IF (ipTcComObj=0) THEN
  GetObjPara := Tc2_System.E_HRESULTAdsErr.NOINTERFACE;
END_IF

IF (SUCCEEDED(GetObjPara)) THEN
  GetObjPara := ipTcComObj.TcGetObjPara(pid:=pid,nData,pData,0);
END_IF
END_METHOD

{attribute 'object_name' := 'Init'}
METHOD PROTECTED Init : HRESULT
VAR_INPUT
	oid: OTCID;
END_VAR

// preinitialize variables
memset(ADR(moduleClsId),0,SIZEOF(moduleClsId));
bClassIdVerified := FALSE;
hResult := Tc2_System.E_HRESULTAdsErr.HRESULT_ADS_NOERROR;

// get object server
IF (ipObjSrv=0) THEN
  hResult := FW_ObjMgr_GetObjectServer(_AppInfo.ObjId,ADR(ipObjSrv));
END_IF

// try to get object interfaces
IF (SUCCEEDED(hresult)) THEN
  QueryTcComInterface(hResult,oid);
END_IF

// verify class id
IF (SUCCEEDED(hresult)) THEN
  hresult := VerifyClassId();
END_IF

// query interfaces, if the current state is higher than INIT
IF (SUCCEEDED(hresult) AND State>TCOM_STATE.TCOM_STATE_INIT) THEN
  QueryObjInterfaces(hResult);
END_IF

// return value
Init := hresult;
END_METHOD

{attribute 'object_name' := 'InitObjName'}
METHOD PRIVATE InitObjName
VAR_INPUT
	hr: REFERENCE TO HRESULT;
END_VAR
VAR
	objectName: STRING(255) := 'TempContr_PlcRtFbInstance';
	oid: OTCID;
END_VAR

IF (SUCCEEDED(hr)) THEN
  hr := ipTcComObj.TcGetObjectId(oid);
END_IF

IF (SUCCEEDED(hr) and bDynInstance) THEN
  objectName := TC2_STANDARD.CONCAT(objectName,'_');
  objectName := TC2_STANDARD.CONCAT(objectName,UDINT_TO_STRING(oid));
  hr := ipTcComObj.TcSetObjectName(ADR(objectName));
END_IF
END_METHOD

{attribute 'object_name' := 'Internal_SetObjState'}
METHOD PROTECTED Internal_SetObjState
VAR_INPUT
	hr: REFERENCE TO HRESULT;
	nextState: TCOM_STATE;
END_VAR

// verify class id
IF (SUCCEEDED(hr)) THEN
  hr := VerifyClassId();
END_IF

// switch object state
IF (SUCCEEDED(hr) AND nextState>=TCOM_STATE_INIT) THEN
  IF (ipTcComObj=0) THEN
    hr := Tc2_System.E_HRESULTAdsErr.NOINTERFACE;
  END_IF
  IF (ipObjSrv=0) THEN
    hr := Tc2_System.E_HRESULTAdsErr.NOINTERFACE;
  END_IF
  IF (SUCCEEDED(hr)) THEN
    hr := ipTcComObj.TcSetObjState(nextState,ipObjSrv,pInitData);
  END_IF
END_IF
END_METHOD

{attribute 'object_name' := 'QueryObjInterface'}
METHOD PRIVATE QueryObjInterface
VAR_INPUT
	hr: REFERENCE TO HRESULT;
	iid: REFERENCE TO IID;
	pipItf: POINTER TO ITcUnknown;
END_VAR
VAR CONSTANT
	pNull: PVOID := 0;
END_VAR

IF (SUCCEEDED(hr)) THEN
  IF (ipTcComObj=0) THEN
    hr := Tc2_System.E_HRESULTAdsErr.NOINTERFACE;
  ELSIF (pipItf^=ULINT_TO_DWORD(pNull)) THEN
    hr := ipTcComObj.TcQueryInterface(iid:= iid, pipItf:=pipItf);
  END_IF
END_IF
END_METHOD

{attribute 'object_name' := 'QueryObjInterfaces'}
METHOD PRIVATE QueryObjInterfaces
VAR_INPUT
	hr: REFERENCE TO HRESULT;
END_VAR

IF(State<TCOM_STATE_PREOP)THEN
  hr := Tc2_System.E_HRESULTAdsErr.INVALIDSTATE;
END_IF

//cyclic interface
QueryObjInterface(hr,IID_ITCCYCLIC,ADR(ipTcCyclic));
//post cyclic interface
QueryObjInterface(hr,IID_ITCPOSTCYCLIC,ADR(ipTcPostCyclic));
//adi interface
QueryObjInterface(hr,IID_ITcADI,ADR(ipTcAdi));
END_METHOD

{attribute 'object_name' := 'QueryTcComInterface'}
METHOD PRIVATE QueryTcComInterface
VAR_INPUT
	hr: REFERENCE TO HRESULT;
	oid: OTCID;
END_VAR

IF (ipObjSrv=0) THEN
  hr := Tc2_System.E_HRESULTAdsErr.NOINTERFACE;
END_IF

IF (SUCCEEDED(hr) AND ipTcComObj=0) THEN
  bDynInstance := FALSE;
  IF(oid>0) THEN
    // query interface of existing object
    hr := ipObjSrv.TcQueryObjectInterface(oid,IID_ITComObject,ADR(ipTcComObj));
  ELSE
    // create new instance and get the object interface
    hr := ipObjSrv.TcCreateInstance(assignedClsId,IID_ITComObject,ADR(ipTcComObj));
    IF (SUCCEEDED(hr)) THEN
      bDynInstance := TRUE;
      hr := ipTcComObj.TcSetObjectId(OTCID_CreateNewId);
    END_IF
  END_IF
  IF (SUCCEEDED(hr)) THEN
    eInitialObjState := State;
  END_IF
END_IF
END_METHOD

{attribute 'object_name' := 'ReadModuleClassId'}
METHOD PRIVATE ReadModuleClassId : HRESULT
VAR
	emptyClsId: CLSID;
END_VAR
memset(ADR(emptyClsId),0,SIZEOF(emptyClsId));
IF (memcmp(ADR(moduleClsId),ADR(emptyClsId),SIZEOF(moduleClsId))=0) THEN
  IF (ipTcComObj=0) THEN
    ReadModuleClassId := Tc2_System.E_HRESULTAdsErr.NOINTERFACE;
  END_IF

  //objectClsId := clsid;
  IF (SUCCEEDED(ReadModuleClassId)) THEN
    ReadModuleClassId := ipTcComObj.GetClassId(moduleClsId);
  END_IF
END_IF
END_METHOD

{attribute 'object_name' := 'ReleaseImagePtrs'}
METHOD PRIVATE ReleaseImagePtrs : HRESULT
VAR
	nDaIdx: UDINT;
	pCurDataArea: POINTER TO ST_TcMatSimObjectDataAreaInfo;
END_VAR

IF (ipTcAdi=0) THEN
  ReleaseImagePtrs := Tc2_System.E_HRESULTAdsErr.NOINTERFACE;
END_IF

IF (SUCCEEDED(ReleaseImagePtrs) AND pDataAreas<>0) THEN
  // release pointers to the simulink module process images
  FOR nDaIdx:=0 TO nDataAreas-1 DO
    pCurDataArea := pDataAreas + nDaIdx*SIZEOF(ST_TcMatSimObjectDataAreaInfo);

    IF (pCurDataArea^.pModuleProcImg<>0) THEN
      ipTcAdi.ReleaseImagePtr(pData:=pCurDataArea^.pModuleProcImg);
      pCurDataArea^.pModuleProcImg := 0;
    END_IF
  END_FOR
END_IF
END_METHOD

{attribute 'object_name' := 'ReleaseObjInterfaces'}
METHOD PRIVATE ReleaseObjInterfaces : HRESULT

// release interface pointers
IF (ipTcCyclic<>0) THEN
  ipTcCyclic.TcRelease();
  ipTcCyclic := 0;
END_IF
IF (ipTcPostCyclic<>0) THEN
  ipTcPostCyclic.TcRelease();
  ipTcPostCyclic := 0;
END_IF
IF (ipTcAdi<>0) THEN
  ipTcAdi.TcRelease();
  ipTcAdi := 0;
END_IF
END_METHOD

{attribute 'object_name' := 'ReleaseTcComInterface'}
METHOD PRIVATE ReleaseTcComInterface : HRESULT
VAR
	nStateChangeCnt: DINT := 0;
END_VAR

IF (ipTcComObj<>0) THEN
  WHILE (State>eInitialObjState AND nStateChangeCnt<1000) DO
    State := eInitialObjState;
    nStateChangeCnt := nStateChangeCnt+1;
  END_WHILE
  ReleaseObjInterfaces();
  IF (bDynInstance) THEN
    ReleaseTcComInterface := TC3_MODULE.FW_ObjMgr_DeleteInstance(ADR(ipTcComObj));
  ELSE
    ipTcComObj.TcRelease();
  END_IF
  ipTcComObj := 0;
END_IF
END_METHOD

{attribute 'object_name' := 'ResetHresult'}
METHOD ResetHresult
hResult := S_OK;
END_METHOD

{attribute 'object_name' := 'SaveOnlineParametersForInit'}
METHOD SaveOnlineParametersForInit : HRESULT
VAR
	idx: UINT;
	pInitElemHdr: POINTER TO TComInitDataElmHdr;
	pData: PVOID;
	nData: UDINT;
END_VAR
VAR CONSTANT
	nInitDataAlignment: UDINT := 4;
END_VAR
IF (pInitData<>0) THEN
  pInitElemHdr := pInitData + SIZEOF(pInitData^);
  FOR idx:=1 TO pInitData^.uiElmCnt DO
    pData := pInitElemHdr + ULINT_TO_DWORD(SIZEOF(pInitElemHdr^));
    nData := pInitElemHdr^.cbData;
    SaveOnlineParametersForInit := GetObjPara(pInitElemHdr^.indexOffset,nData,pData);
    IF (FAILED(SaveOnlineParametersForInit)) THEN
      RETURN;
    END_IF
    pInitElemHdr := pData + (nInitDataAlignment*((nData + nInitDataAlignment - 1)/nInitDataAlignment));
  END_FOR
ELSE
	SaveOnlineParametersForInit := Tc2_System.E_HRESULTAdsErr.NOTINIT;
END_IF
END_METHOD


METHOD PUBLIC SetDataAreaInfo
VAR_INPUT
  pDataAreas: POINTER TO ST_TcMatSimObjectDataAreaInfo;
  nDataAreas: UDINT;
END_VAR

THIS^.nDataAreas := nDataAreas;
THIS^.pDataAreas := pDataAreas;
END_METHOD


METHOD PUBLIC SetInitDataInfo
VAR_INPUT
  pInitData : POINTER TO TComInitDataHdr;
END_VAR
this^.pInitData := pInitData;
END_METHOD

{attribute 'object_name' := 'SetObjPara'}
METHOD SetObjPara : HRESULT
VAR_INPUT
	pid: PTCID;
	nData: UDINT;
	pData: PVOID;
END_VAR

IF (ipTcComObj=0) THEN
  SetObjPara := Tc2_System.E_HRESULTAdsErr.NOINTERFACE;
END_IF

IF (SUCCEEDED(SetObjPara)) THEN
  SetObjPara := ipTcComObj.TcSetObjPara(pid:=pid,nData,pData,0);
END_IF
END_METHOD

{attribute 'object_name' := 'SetObjState'}
METHOD SetObjState : HRESULT
VAR_INPUT
	finalState: TCOM_STATE;
END_VAR
VAR
	bShiftUp: BOOL;
	bShiftDown: BOOL;
	currentState: TCOM_STATE;
END_VAR

currentState := State;

bShiftUp := finalState>currentState;
bShiftDown := finalState<currentState;

// do not switch up on error
IF (FAILED(hresult)) THEN
  bShiftUp := FALSE;
END_IF
// reset existing error on switching down
IF (bShiftDown) THEN
  ResetHresult();
END_IF

// prepared state switch
CASE currentState OF
  TCOM_STATE_INIT:
    IF(bShiftUp) THEN
      QueryTcComInterface(hResult,0);
      Internal_SetObjState(hResult,TCOM_STATE.TCOM_STATE_PREOP);
      InitObjName(hResult);
    END_IF

  TCOM_STATE_PREOP:
    IF(bShiftUp) THEN
      Internal_SetObjState(hResult,TCOM_STATE.TCOM_STATE_SAFEOP);
      QueryObjInterfaces(hResult);
    ELSIF (bShiftDown) THEN
      Internal_SetObjState(hResult,TCOM_STATE.TCOM_STATE_INIT);
    END_IF

  TCOM_STATE_SAFEOP:
    IF(bShiftUp) THEN
      Internal_SetObjState(hResult,TCOM_STATE.TCOM_STATE_OP);
      QueryObjInterfaces(hResult);
    ELSIF (bShiftDown) THEN
      Internal_SetObjState(hResult,TCOM_STATE.TCOM_STATE_PREOP);
      ReleaseObjInterfaces();
    END_IF


  TCOM_STATE_OP:
    IF (bShiftDown) THEN
      Internal_SetObjState(hResult,TCOM_STATE.TCOM_STATE_SAFEOP);
    END_IF
END_CASE

SetObjState := hResult;
END_METHOD

PROPERTY State : TCOM_STATE
GET
VAR
	hr: HRESULT := S_OK;
	eObjState: TCOM_STATE;
END_VAR

IF (ipTcComObj<>0) THEN
  hr := ipTcComObj.TcGetObjState(ADR(eObjState));
IF (FAILED(hr)) THEN
  eObjState := TCOM_STATE.TCOM_STATE_INIT;
END_IF
ELSE
  eObjState := TCOM_STATE.TCOM_STATE_INIT;
END_IF
State := eObjState;
END_GET
SET
SetObjState(State);
END_SET
END_PROPERTY

{attribute 'object_name' := 'VerifyClassId'}
METHOD PRIVATE VerifyClassId : HRESULT
VAR
	emptyClsId: CLSID;
END_VAR
memset(ADR(emptyClsId),0,SIZEOF(emptyClsId));
IF (bClassIdVerified) THEN
  // class ID was already verified
  VerifyClassId := Tc2_System.E_HRESULTAdsErr.HRESULT_ADS_NOERROR;
ELSIF (memcmp(ADR(assignedClsId),ADR(emptyClsId),SIZEOF(assignedClsId))=0) THEN
  // skip class ID verification if no assignedClsId specified
  VerifyClassId := Tc2_System.E_HRESULTAdsErr.HRESULT_ADS_NOERROR;
ELSE
  // verify class ID
  VerifyClassId := ReadModuleClassId();

  IF (SUCCEEDED(VerifyClassId)) THEN
    IF (memcmp(ADR(assignedClsId),ADR(moduleClsId),SIZEOF(assignedClsId))<>0) THEN
     VerifyClassId := Tc2_System.E_HRESULTAdsErr.INVALIDCLSID;
    END_IF
  END_IF
  bClassIdVerified := SUCCEEDED(VerifyClassId);
END_IF
END_METHOD

END_FUNCTION_BLOCK

// ---- GlobalTextList.TcGTLO
TEXTLIST GlobalTextList
  145 = ' %.2f'
  175 = ' realState=%.3f'
  165 = ' t_Interval=%.2f'
  167 = ' t_Interval=%.3f'
  169 = ' t_Interval=%.4f'
  168 = ' t_Interval=%.5f'
  143 = '%.2f'
  179 = '1'
  81 = 'Axis10_Back'
  82 = 'Axis10_Home'
  117 = 'Axis10_Move'
  11 = 'Axis10_Power'
  83 = 'Axis11_Back'
  84 = 'Axis11_Home'
  118 = 'Axis11_Move'
  12 = 'Axis11_Power'
  85 = 'Axis12_Back'
  86 = 'Axis12_Home'
  119 = 'Axis12_Move'
  13 = 'Axis12_Power'
  87 = 'Axis13_Back'
  88 = 'Axis13_Home'
  120 = 'Axis13_Move'
  14 = 'Axis13_Power'
  89 = 'Axis14_Back'
  90 = 'Axis14_Home'
  121 = 'Axis14_Move'
  15 = 'Axis14_Power'
  91 = 'Axis15_Back'
  92 = 'Axis15_Home'
  122 = 'Axis15_Move'
  16 = 'Axis15_Power'
  93 = 'Axis16_Back'
  94 = 'Axis16_Home'
  123 = 'Axis16_Move'
  17 = 'Axis16_Power'
  95 = 'Axis17_Back'
  96 = 'Axis17_Home'
  124 = 'Axis17_Move'
  18 = 'Axis17_Power'
  97 = 'Axis18_Back'
  98 = 'Axis18_Home'
  125 = 'Axis18_Move'
  19 = 'Axis18_Power'
  62 = 'Axis1_Back'
  64 = 'Axis1_Home'
  63 = 'Axis1_Home_Set'
  106 = 'Axis1_M'
  108 = 'Axis1_Move'
  2 = 'Axis1_Power'
  65 = 'Axis2_Back'
  66 = 'Axis2_Home'
  109 = 'Axis2_Move'
  3 = 'Axis2_Power'
  67 = 'Axis3_Back'
  68 = 'Axis3_Home'
  110 = 'Axis3_Move'
  4 = 'Axis3_Power'
  69 = 'Axis4_Back'
  70 = 'Axis4_Home'
  111 = 'Axis4_Move'
  5 = 'Axis4_Power'
  71 = 'Axis5_Back'
  72 = 'Axis5_Home'
  112 = 'Axis5_Move'
  6 = 'Axis5_Power'
  73 = 'Axis6_Back'
  74 = 'Axis6_Home'
  113 = 'Axis6_Move'
  7 = 'Axis6_Power'
  75 = 'Axis7_Back'
  76 = 'Axis7_Home'
  114 = 'Axis7_Move'
  8 = 'Axis7_Power'
  77 = 'Axis8_Back'
  78 = 'Axis8_Home'
  115 = 'Axis8_Move'
  9 = 'Axis8_Power'
  79 = 'Axis9_Back'
  80 = 'Axis9_Home'
  116 = 'Axis9_Move'
  10 = 'Axis9_Power'
  56 = 'Axis_ActPostion[INDEX]'
  60 = 'Back'
  174 = 'Botton For Step'
  57 = 'Current_Turque_Value[INDEX]'
  39 = 'Driver10_Reset'
  40 = 'Driver11_Reset'
  41 = 'Driver12_Reset'
  42 = 'Driver13_Reset'
  43 = 'Driver14_Reset'
  44 = 'Driver15_Reset'
  45 = 'Driver16_Reset'
  46 = 'Driver17_Reset'
  47 = 'Driver18_Reset'
  30 = 'Driver1_Reset'
  31 = 'Driver2_Reset'
  32 = 'Driver3_Reset'
  33 = 'Driver4_Reset'
  34 = 'Driver5_Reset'
  35 = 'Driver6_Reset'
  36 = 'Driver7_Reset'
  37 = 'Driver8_Reset'
  38 = 'Driver9_Reset'
  127 = 'Error & Reset'
  126 = 'Error&Reset'
  151 = 'Exsetopint_Enable'
  152 = 'Exsetopint_On'
  141 = 'Exsetpoint_Exectue'
  23 = 'Home'
  59 = 'Home_Execute'
  61 = 'Home_Set'
  131 = 'Leg1_Home'
  181 = 'Leg21'
  132 = 'Leg2_Home'
  133 = 'Leg3_Home'
  134 = 'Leg4_Home'
  135 = 'Leg5_Home'
  136 = 'Leg6_Home'
  180 = 'Leg_1'
  186 = 'Leg_16'
  182 = 'Leg_2'
  183 = 'Leg_3'
  184 = 'Leg_4'
  185 = 'Leg_5'
  187 = 'Leg_6'
  177 = 'Model_Position[INDEX]'
  130 = 'Move & Stand'
  107 = 'MoveAbsoluteDone[INDEX]'
  129 = 'Move_Execute'
  53 = 'Power'
  20 = 'Power_Execute'
  188 = 'RealState=%.3f'
  29 = 'Reset'
  49 = 'Reset_Execute'
  26 = 'Robot_Error'
  101 = 'Robot_Home_Set'
  0 = 'Robot_Power'
  48 = 'Robot_Reset'
  128 = 'Robot_Stand_Execute'
  99 = 'Robot_Start_Back'
  100 = 'sadad'
  166 = 'Simulink_Move'
  176 = 'State=%.3f'
  189 = 'Step_Test'
  147 = 't=%.2f'
  170 = 't=%.3f'
  171 = 'Touch_Signal'
  178 = 'Touch_Signal(模型中腿编号)'
  172 = 'Touch_Signal_1'
  173 = 'Touch_Signal_Change'
  144 = 'T_ALL = %.2f'
  158 = 't_Interval=%.2f'
  22 = '切换视图'
  157 = '取样时间间隔 t_Interval'
  160 = '取样时间间隔 t_Interval(ms)'
  161 = '取样时间间隔 t_Interval(s)'
  159 = '取样时间间隔 t_Interval/ms'
  139 = '可以用来整体机器人运动'
  140 = '可以用来整体机器人进行Simulink模型验证'
  104 = '可以用来给单个四缸伸长或者是整体机器人站立'
  28 = '可以用来给单个电机或者是整体机器人上电'
  55 = '可以用来给单个电机或者是整体机器人找零'
  103 = '可以用来给单个电机或者是整体机器人站立'
  52 = '可以用来错误时给单个电机或者是整体机器人进行驱动重置'
  24 = '否'
  149 = '开始输入轨迹'
  156 = '当前取样时间 t'
  163 = '当前取样时间 t(s)'
  25 = '是'
  148 = '是否开始输入轨迹'
  21 = '是否进行上电操作'
  58 = '是否进行找零操作'
  1 = '是否进行整机操作'
  142 = '是否进行运动操作'
  50 = '是否进行驱动重置'
  138 = '本界面为电机Sumulink模型运动程序：'
  137 = '本界面为电机Sumulink程序：'
  27 = '本界面为电机上电程序：'
  102 = '本界面为电机伸长/机器人站立程序：'
  54 = '本界面为电机找零程序：'
  105 = '本界面为电机绝对运动/机器人站立程序：'
  51 = '本界面为驱动重置程序：'
  154 = '输入运动总时长 T_ALL'
  162 = '输入运动总时长 T_ALL(s)'
  150 = '运动当前时间 t'
  164 = '运动当前时间 t(s)'
  146 = '运动总时长 T_ALL'
  155 = '运动时间间隔 t'
  153 = '运动终止信号'
END_TEXTLIST

// ---- VISUs/Visu_Home.TcVIS
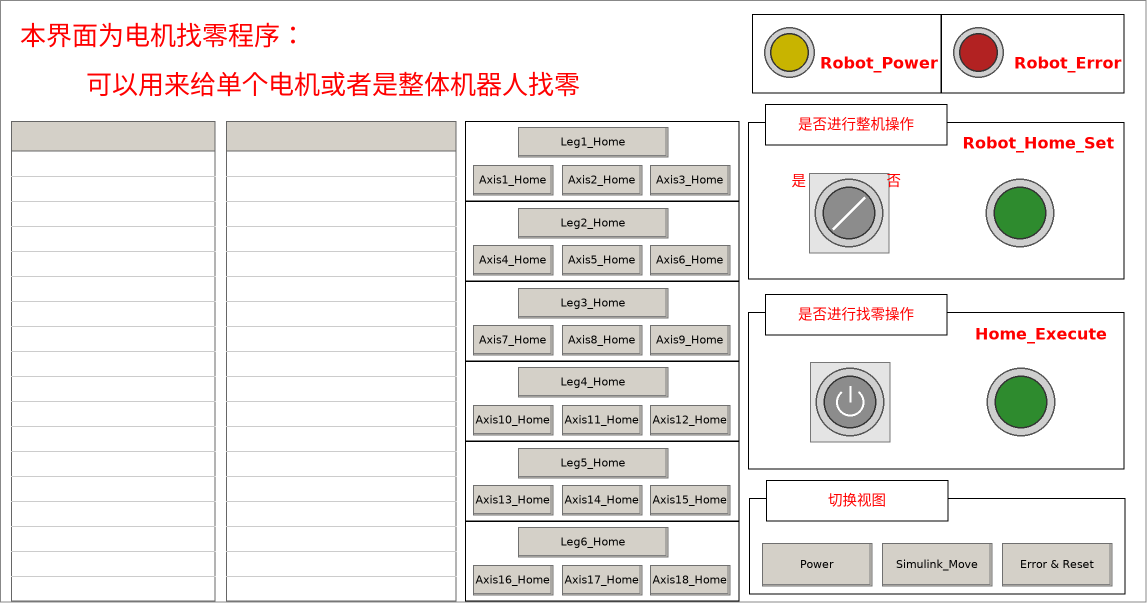
VISUALIZATION Visu_Home  // 1147x603
    Rectangle (752,14 189x79)
    Rectangle (748,312 376x157)
    Label (964,318 154x32), "Home_Execute"
    Rectangle (765,294 182x41), "是否进行找零操作"
    Lamp1 (981,362 80x80), variable: MAIN.Home_Execute, style: Lamp-Lamp1-Green
    PowerSwitch (810,362 80x80), variable: MAIN.Home_Execute, behaviour: TOGGLE, style: Switch-PowerSwitch-Gray
    Rectangle (941,14 183x79)
    Lamp1 (948,23 61x59), variable: MAIN.Robot_Error, style: Lamp-Lamp1-Red
    Label (991,47 154x32), "Robot_Error"
    Label (17,15 365x42), "本界面为电机找零程序："
    Label (83,64 874x42), "可以用来给单个电机或者是整体机器人找零"
    Table (11,121 204x480), data array: MAIN.Axis_ActPostion
        p3854506369: MAIN.Axis_ActPostion[INDEX]
    Table (226,121 230x480), data array: MAIN.Current_Turque_Value
        p3854506369: MAIN.Current_Turque_Value[INDEX]
    Lamp1 (759,23 61x59), variable: MAIN.Robot_Power, style: Lamp-Lamp1-Yellow
    Label (802,47 154x32), "Robot_Power"
    Rectangle (465,121 274x80)
    Button (473,165 80x30), "Axis1_Home"
        toggle MAIN.Axis_Home_Set[1]
        OnMouseClick: change screen: Visu_Home
    Button (650,165 80x30), "Axis3_Home"
        toggle MAIN.Axis_Home_Set[3]
        OnMouseClick: change screen: Visu_Home
    Button (562,165 80x30), "Axis2_Home"
        toggle MAIN.Axis_Home_Set[2]
        OnMouseClick: change screen: Visu_Home
    Rectangle (465,201 274x80)
    Button (473,245 80x30), "Axis4_Home"
        toggle MAIN.Axis_Home_Set[4]
        OnMouseClick: change screen: Visu_Home
    Button (650,245 80x30), "Axis6_Home"
        toggle MAIN.Axis_Home_Set[6]
        OnMouseClick: change screen: Visu_Home
    Button (562,245 80x30), "Axis5_Home"
        toggle MAIN.Axis_Home_Set[5]
        OnMouseClick: change screen: Visu_Home
    Rectangle (465,281 274x80)
    Button (473,325 80x30), "Axis7_Home"
        toggle MAIN.Axis_Home_Set[7]
        OnMouseClick: change screen: Visu_Home
    Button (650,325 80x30), "Axis9_Home"
        toggle MAIN.Axis_Home_Set[9]
        OnMouseClick: change screen: Visu_Home
    Button (562,325 80x30), "Axis8_Home"
        toggle MAIN.Axis_Home_Set[8]
        OnMouseClick: change screen: Visu_Home
    Rectangle (465,361 274x80)
    Button (473,405 80x30), "Axis10_Home"
        toggle MAIN.Axis_Home_Set[10]
        OnMouseClick: change screen: Visu_Home
    Button (650,405 80x30), "Axis12_Home"
        toggle MAIN.Axis_Home_Set[12]
        OnMouseClick: change screen: Visu_Home
    Button (562,405 80x30), "Axis11_Home"
        toggle MAIN.Axis_Home_Set[11]
        OnMouseClick: change screen: Visu_Home
    Rectangle (465,441 274x80)
    Button (473,485 80x30), "Axis13_Home"
        toggle MAIN.Axis_Home_Set[13]
        OnMouseClick: change screen: Visu_Home
    Button (650,485 80x30), "Axis15_Home"
        toggle MAIN.Axis_Home_Set[15]
        OnMouseClick: change screen: Visu_Home
    Button (562,485 80x30), "Axis14_Home"
        toggle MAIN.Axis_Home_Set[14]
        OnMouseClick: change screen: Visu_Home
    Rectangle (465,521 274x80)
    Button (473,565 80x30), "Axis16_Home"
        toggle MAIN.Axis_Home_Set[16]
        OnMouseClick: change screen: Visu_Home
    Button (650,565 80x30), "Axis18_Home"
        toggle MAIN.Axis_Home_Set[18]
        OnMouseClick: change screen: Visu_Home
    Button (562,565 80x30), "Axis17_Home"
        toggle MAIN.Axis_Home_Set[17]
        OnMouseClick: change screen: Visu_Home
    Rectangle (749,498 376x96)
    Rectangle (766,480 182x41), "切换视图"
    Button (762,543 110x43), "Power"
        OnMouseClick: change screen: Visu_Power
    Button (1002,543 110x43), "Error & Reset"
        OnMouseClick: change screen: Visu_Reset
    Button (882,543 110x43), "Simulink_Move"
        OnMouseClick: change screen: Visu_SimulinkMove
    Rectangle (748,122 376x157)
    Rectangle (765,104 182x41), "是否进行整机操作"
    Lamp1 (980,173 80x80), variable: MAIN.Robot_Home_Set, style: Lamp-Lamp1-Green
    RotarySwitch (809,173 80x80), variable: MAIN.Robot_Home_Set, behaviour: TOGGLE, style: Switch-RotarySwitch-Gray
    Label (864,166 60x30), "否"
    Label (769,166 60x30), "是"
    Label (935,127 207x32), "Robot_Home_Set"
    Button (518,127 150x30), "Leg1_Home"
        tap MAIN.Leg_Home_Set[1]
    Button (518,208 150x30), "Leg2_Home"
        tap MAIN.Leg_Home_Set[2]
    Button (518,288 150x30), "Leg3_Home"
        tap MAIN.Leg_Home_Set[3]
    Button (518,367 150x30), "Leg4_Home"
        tap MAIN.Leg_Home_Set[4]
    Button (518,448 150x30), "Leg5_Home"
        tap MAIN.Leg_Home_Set[5]
    Button (518,527 150x30), "Leg6_Home"
        tap MAIN.Leg_Home_Set[6]
END_VISUALIZATION

// ---- VISUs/Visu_Power.TcVIS
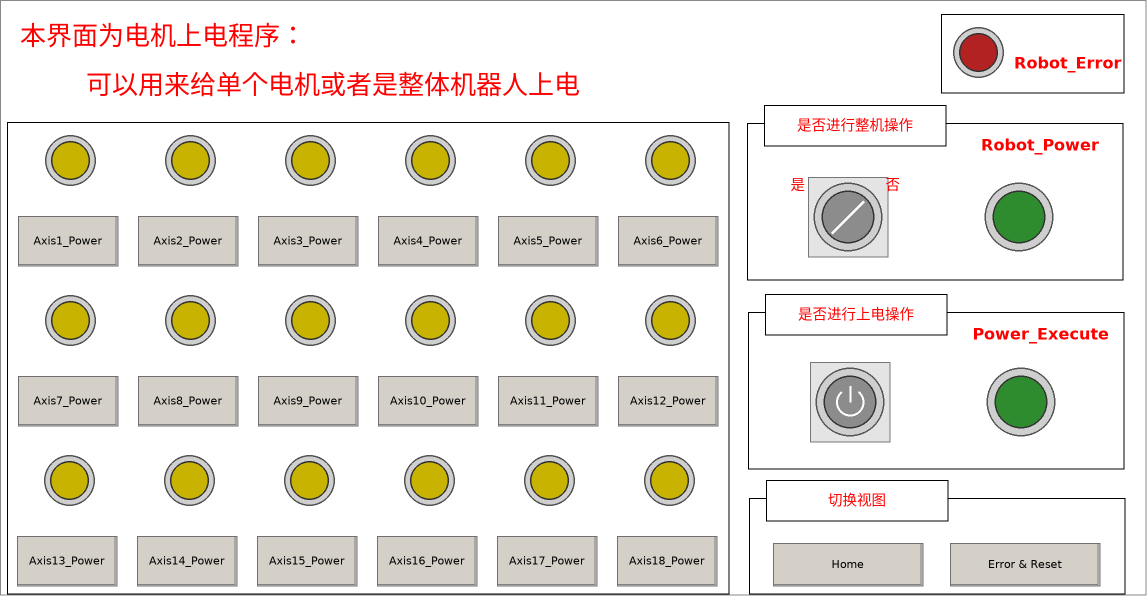
VISUALIZATION Visu_Power  // 1147x596
    Label (987,37 154x32), "Robot_Error"
    Rectangle (7,122 722x472)
    Lamp1 (40,131 61x59), variable: MAIN.Power_Status[1], style: Lamp-Lamp1-Yellow
    Lamp1 (160,131 61x59), variable: MAIN.Power_Status[2], style: Lamp-Lamp1-Yellow
    Lamp1 (280,131 61x59), variable: MAIN.Power_Status[3], style: Lamp-Lamp1-Yellow
    Lamp1 (400,131 61x59), variable: MAIN.Power_Status[4], style: Lamp-Lamp1-Yellow
    Lamp1 (520,131 61x59), variable: MAIN.Power_Status[5], style: Lamp-Lamp1-Yellow
    Lamp1 (640,131 61x59), variable: MAIN.Power_Status[6], style: Lamp-Lamp1-Yellow
    Button (18,216 100x50), "Axis1_Power"
        toggle MAIN.Axis_Power[1]
    Button (138,216 100x50), "Axis2_Power"
        toggle MAIN.Axis_Power[2]
    Button (258,216 100x50), "Axis3_Power"
        toggle MAIN.Axis_Power[3]
    Button (378,216 100x50), "Axis4_Power"
        toggle MAIN.Axis_Power[4]
    Button (498,216 100x50), "Axis5_Power"
        toggle MAIN.Axis_Power[5]
    Button (618,216 100x50), "Axis6_Power"
        toggle MAIN.Axis_Power[6]
    Lamp1 (40,291 61x59), variable: MAIN.Power_Status[7], style: Lamp-Lamp1-Yellow
    Lamp1 (160,291 61x59), variable: MAIN.Power_Status[8], style: Lamp-Lamp1-Yellow
    Lamp1 (280,291 61x59), variable: MAIN.Power_Status[9], style: Lamp-Lamp1-Yellow
    Lamp1 (400,291 61x59), variable: MAIN.Power_Status[10], style: Lamp-Lamp1-Yellow
    Lamp1 (520,291 61x59), variable: MAIN.Power_Status[11], style: Lamp-Lamp1-Yellow
    Lamp1 (640,291 61x59), variable: MAIN.Power_Status[12], style: Lamp-Lamp1-Yellow
    Button (18,376 100x50), "Axis7_Power"
        toggle MAIN.Axis_Power[7]
    Button (138,376 100x50), "Axis8_Power"
        toggle MAIN.Axis_Power[8]
    Button (258,376 100x50), "Axis9_Power"
        toggle MAIN.Axis_Power[9]
    Button (378,376 100x50), "Axis10_Power"
        toggle MAIN.Axis_Power[10]
    Button (498,376 100x50), "Axis11_Power"
        toggle MAIN.Axis_Power[11]
    Button (618,376 100x50), "Axis12_Power"
        toggle MAIN.Axis_Power[12]
    Lamp1 (39,451 61x59), variable: MAIN.Power_Status[13], style: Lamp-Lamp1-Yellow
    Lamp1 (159,451 61x59), variable: MAIN.Power_Status[14], style: Lamp-Lamp1-Yellow
    Lamp1 (279,451 61x59), variable: MAIN.Power_Status[15], style: Lamp-Lamp1-Yellow
    Lamp1 (399,451 61x59), variable: MAIN.Power_Status[16], style: Lamp-Lamp1-Yellow
    Lamp1 (519,451 61x59), variable: MAIN.Power_Status[17], style: Lamp-Lamp1-Yellow
    Lamp1 (639,451 61x59), variable: MAIN.Power_Status[18], style: Lamp-Lamp1-Yellow
    Button (17,536 100x50), "Axis13_Power"
        toggle MAIN.Axis_Power[13]
    Button (137,536 100x50), "Axis14_Power"
        toggle MAIN.Axis_Power[14]
    Button (257,536 100x50), "Axis15_Power"
        toggle MAIN.Axis_Power[15]
    Button (377,536 100x50), "Axis16_Power"
        toggle MAIN.Axis_Power[16]
    Button (497,536 100x50), "Axis17_Power"
        toggle MAIN.Axis_Power[17]
    Button (617,536 100x50), "Axis18_Power"
        toggle MAIN.Axis_Power[18]
    Rectangle (748,312 376x157)
    Label (964,318 154x32), "Power_Execute"
    Rectangle (765,294 182x41), "是否进行上电操作"
    Lamp1 (981,362 80x80), variable: MAIN.Power_Execute, style: Lamp-Lamp1-Green
    Rectangle (749,498 376x96)
    Rectangle (766,480 182x41), "切换视图"
    Button (773,543 150x43), "Home"
        OnMouseClick: change screen: Visu_Home
    PowerSwitch (810,362 80x80), variable: MAIN.Power_Execute, behaviour: TOGGLE, style: Switch-PowerSwitch-Gray
    Rectangle (941,14 183x79)
    Lamp1 (948,23 61x59), variable: MAIN.Robot_Error, style: Lamp-Lamp1-Red
    Label (17,15 365x42), "本界面为电机上电程序："
    Label (83,64 639x42), "可以用来给单个电机或者是整体机器人上电"
    Button (950,543 150x43), "Error & Reset"
        OnMouseClick: change screen: Visu_Reset
    Rectangle (747,123 376x157)
    Label (963,129 154x32), "Robot_Power"
    Rectangle (764,105 182x41), "是否进行整机操作"
    Lamp1 (979,177 80x80), variable: MAIN.Robot_Power, style: Lamp-Lamp1-Green
    RotarySwitch (808,177 80x80), variable: MAIN.Robot_Power, behaviour: TOGGLE, style: Switch-RotarySwitch-Gray
    Label (863,170 60x30), "否"
    Label (768,170 60x30), "是"
    Label (991,47 154x32), "Robot_Error"
END_VISUALIZATION

// ---- VISUs/Visu_Reset.TcVIS
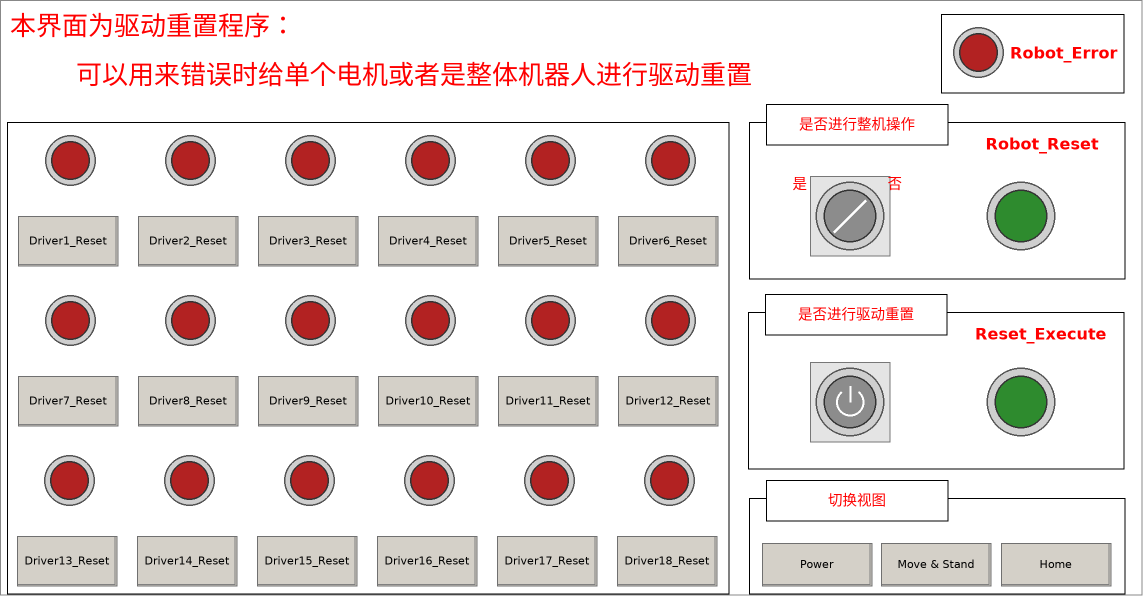
VISUALIZATION Visu_Reset  // 1143x596
    Rectangle (7,122 722x472)
    Lamp1 (40,131 61x59), variable: MAIN.Axis_Error[1], style: Lamp-Lamp1-Red
    Lamp1 (160,131 61x59), variable: MAIN.Axis_Error[2], style: Lamp-Lamp1-Red
    Lamp1 (280,131 61x59), variable: MAIN.Axis_Error[3], style: Lamp-Lamp1-Red
    Lamp1 (400,131 61x59), variable: MAIN.Axis_Error[4], style: Lamp-Lamp1-Red
    Lamp1 (520,131 61x59), variable: MAIN.Axis_Error[5], style: Lamp-Lamp1-Red
    Lamp1 (640,131 61x59), variable: MAIN.Axis_Error[6], style: Lamp-Lamp1-Red
    Button (18,216 100x50), "Driver1_Reset"
        tap MAIN.Axis_Reset[1]
    Button (138,216 100x50), "Driver2_Reset"
        tap MAIN.Axis_Reset[2]
    Button (258,216 100x50), "Driver3_Reset"
        tap MAIN.Axis_Reset[3]
    Button (378,216 100x50), "Driver4_Reset"
        tap MAIN.Axis_Reset[4]
    Button (498,216 100x50), "Driver5_Reset"
        tap MAIN.Axis_Reset[5]
    Button (618,216 100x50), "Driver6_Reset"
        tap MAIN.Axis_Reset[6]
    Lamp1 (40,291 61x59), variable: MAIN.Axis_Error[7], style: Lamp-Lamp1-Red
    Lamp1 (160,291 61x59), variable: MAIN.Axis_Error[8], style: Lamp-Lamp1-Red
    Lamp1 (280,291 61x59), variable: MAIN.Axis_Error[9], style: Lamp-Lamp1-Red
    Lamp1 (400,291 61x59), variable: MAIN.Axis_Error[10], style: Lamp-Lamp1-Red
    Lamp1 (520,291 61x59), variable: MAIN.Axis_Error[11], style: Lamp-Lamp1-Red
    Lamp1 (640,291 61x59), variable: MAIN.Axis_Error[12], style: Lamp-Lamp1-Red
    Button (18,376 100x50), "Driver7_Reset"
        tap MAIN.Axis_Reset[7]
    Button (138,376 100x50), "Driver8_Reset"
        tap MAIN.Axis_Reset[8]
    Button (258,376 100x50), "Driver9_Reset"
        tap MAIN.Axis_Reset[9]
    Button (378,376 100x50), "Driver10_Reset"
        tap MAIN.Axis_Reset[10]
    Button (498,376 100x50), "Driver11_Reset"
        tap MAIN.Axis_Reset[11]
    Button (618,376 100x50), "Driver12_Reset"
        tap MAIN.Axis_Reset[12]
    Lamp1 (39,451 61x59), variable: MAIN.Axis_Error[13], style: Lamp-Lamp1-Red
    Lamp1 (159,451 61x59), variable: MAIN.Axis_Error[14], style: Lamp-Lamp1-Red
    Lamp1 (279,451 61x59), variable: MAIN.Axis_Error[15], style: Lamp-Lamp1-Red
    Lamp1 (399,451 61x59), variable: MAIN.Axis_Error[16], style: Lamp-Lamp1-Red
    Lamp1 (519,451 61x59), variable: MAIN.Axis_Error[17], style: Lamp-Lamp1-Red
    Lamp1 (639,451 61x59), variable: MAIN.Axis_Error[18], style: Lamp-Lamp1-Red
    Button (17,536 100x50), "Driver13_Reset"
        tap MAIN.Axis_Reset[13]
    Button (137,536 100x50), "Driver14_Reset"
        tap MAIN.Axis_Reset[14]
    Button (257,536 100x50), "Driver15_Reset"
        tap MAIN.Axis_Reset[15]
    Button (377,536 100x50), "Driver16_Reset"
        tap MAIN.Axis_Reset[16]
    Button (497,536 100x50), "Driver17_Reset"
        tap MAIN.Axis_Reset[17]
    Button (617,536 100x50), "Driver18_Reset"
        tap MAIN.Axis_Reset[18]
    Rectangle (749,122 376x157)
    Label (965,128 154x32), "Robot_Reset"
    Rectangle (766,104 182x41), "是否进行整机操作"
    Rectangle (748,312 376x157)
    Label (964,318 154x32), "Reset_Execute"
    Rectangle (765,294 182x41), "是否进行驱动重置"
    Lamp1 (981,176 80x80), variable: MAIN.Robot_Reset, style: Lamp-Lamp1-Green
    Lamp1 (981,362 80x80), variable: MAIN.Reset_Execute, style: Lamp-Lamp1-Green
    RotarySwitch (810,176 80x80), variable: MAIN.Robot_Reset, behaviour: TOGGLE, style: Switch-RotarySwitch-Gray
    Rectangle (749,498 376x96)
    Rectangle (766,480 182x41), "切换视图"
    Label (865,169 60x30), "否"
    Label (770,169 60x30), "是"
    PowerSwitch (810,362 80x80), variable: MAIN.Reset_Execute, behaviour: TOGGLE, style: Switch-PowerSwitch-Gray
    Label (7,5 365x42), "本界面为驱动重置程序："
    Label (73,54 874x42), "可以用来错误时给单个电机或者是整体机器人进行驱动重置"
    Rectangle (941,14 183x79)
    Lamp1 (948,23 61x59), variable: MAIN.Robot_Error, style: Lamp-Lamp1-Red
    Label (987,37 154x32), "Robot_Error"
    Button (762,543 110x43), "Power"
        OnMouseClick: change screen: Visu_Power
    Button (1001,543 110x43), "Home"
        OnMouseClick: change screen: Visu_Home
    Button (881,543 110x43), "Move & Stand"
        OnMouseClick: change screen: Visu_Stand
END_VISUALIZATION

// ---- VISUs/Visu_SimulinkMove.TcVIS
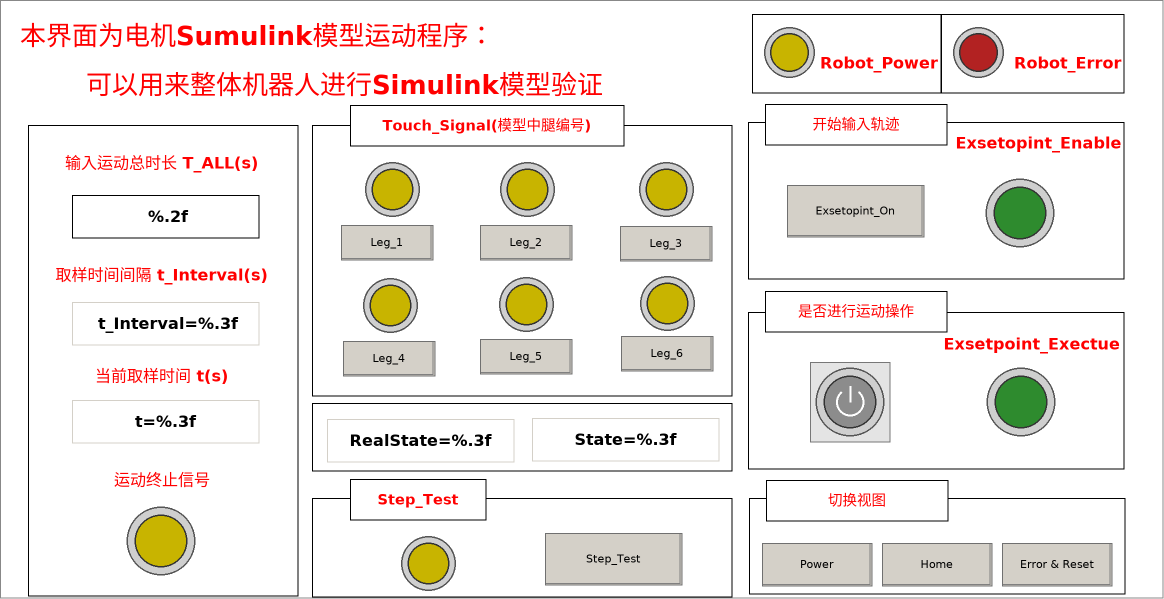
VISUALIZATION Visu_SimulinkMove  // 1164x599
    Rectangle (312,498 420x99)
    Rectangle (749,498 376x96)
    Rectangle (766,480 182x41), "切换视图"
    Button (762,543 110x43), "Power"
        OnMouseClick: change screen: Visu_Power
    Button (1002,543 110x43), "Error & Reset"
        OnMouseClick: change screen: Visu_Reset
    Button (882,543 110x43), "Home"
        OnMouseClick: change screen: Visu_Home
    Rectangle (28,125 270x471)
    Rectangle (752,14 189x79)
    Rectangle (748,312 376x157)
    Label (902,328 260x32), "Exsetpoint_Exectue"
    Rectangle (765,291 182x41), "是否进行运动操作"
    Lamp1 (981,362 80x80), variable: Robot_Movement.ExSetPoint_Execute, style: Lamp-Lamp1-Green
    PowerSwitch (810,362 80x80), variable: Robot_Movement.ExSetPoint_Execute, behaviour: TOGGLE, style: Switch-PowerSwitch-Gray
    Rectangle (941,14 183x79)
    Lamp1 (948,23 61x59), variable: MAIN.Robot_Error, style: Lamp-Lamp1-Red
    Label (991,47 154x32), "Robot_Error"
    Label (17,15 572x42), "本界面为电机Sumulink模型运动程序："
    Label (83,64 874x42), "可以用来整体机器人进行Simulink模型验证"
    Lamp1 (759,23 61x59), variable: MAIN.Robot_Power, style: Lamp-Lamp1-Yellow
    Label (802,47 154x32), "Robot_Power"
    Rectangle (748,122 376x157)
    Rectangle (765,104 182x41), "开始输入轨迹"
    Lamp1 (980,173 80x80), variable: Robot_Movement.ExtSetPointEnable, style: Lamp-Lamp1-Green
    Label (935,127 207x32), "Exsetopint_Enable"
    Rectangle (72,195 187x43), "%.2f", text variable: Robot_Movement.T_All
        OnMouseClick: write Robot_Movement.T_ALL via Default
    Label (32,147 260x32), "输入运动总时长 T_ALL(s)"
    Textfield (72,400 187x43), "t=%.3f", text variable: Robot_Movement.t
    Label (32,360 260x32), "当前取样时间 t(s)"
    Button (787,185 137x52), "Exsetopint_On"
        toggle Robot_Movement.ExtSetPointEnable
    Lamp1 (121,501 80x80), variable: Robot_Movement.ExtSetPointDisable, style: Lamp-Lamp1-Yellow
    Label (32,464 260x32), "运动终止信号"
    Label (32,259 260x32), "取样时间间隔 t_Interval(s)"
    Textfield (72,302 187x43), "t_Interval=%.3f", text variable: Robot_Movement.t_Interval
        OnMouseClick: write Robot_Movement.t_Interval via Default
    Rectangle (312,125 420x271)
    Rectangle (350,105 274x41), "Touch_Signal(模型中腿编号)"
    Lamp1 (361,157 63x65), variable: Robot_Movement.Touch_Signal[1], style: Lamp-Lamp1-Yellow
    Lamp1 (496,157 63x65), variable: Robot_Movement.Touch_Signal[2], style: Lamp-Lamp1-Yellow
    Lamp1 (635,157 63x65), variable: Robot_Movement.Touch_Signal[3], style: Lamp-Lamp1-Yellow
    Lamp1 (359,273 63x65), variable: Robot_Movement.Touch_Signal[4], style: Lamp-Lamp1-Yellow
    Lamp1 (495,272 63x65), variable: Robot_Movement.Touch_Signal[5], style: Lamp-Lamp1-Yellow
    Lamp1 (636,271 63x65), variable: Robot_Movement.Touch_Signal[6], style: Lamp-Lamp1-Yellow
    Rectangle (312,403 420x68)
    Textfield (327,419 187x43), "RealState=%.3f", text variable: Robot_Movement.realState
    Textfield (532,418 187x43), "State=%.3f", text variable: Robot_Movement.state
    Button (545,533 137x52), "Step_Test"
        toggle Robot_Movement.Step_Test
    Lamp1 (397,531 63x65), variable: Robot_Movement.Step_Test, style: Lamp-Lamp1-Yellow
    Rectangle (350,479 136x41), "Step_Test"
    Button (341,225 92x35), "Leg_1"
        toggle Robot_Movement.Touch_Signal[1]
    Button (480,225 92x35), "Leg_2"
        toggle Robot_Movement.Touch_Signal[2]
    Button (620,226 92x35), "Leg_3"
        toggle Robot_Movement.Touch_Signal[3]
    Button (343,341 92x35), "Leg_4"
        toggle Robot_Movement.Touch_Signal[4]
    Button (480,339 92x35), "Leg_5"
        toggle Robot_Movement.Touch_Signal[5]
    Button (621,336 92x35), "Leg_6"
        toggle Robot_Movement.Touch_Signal[6]
END_VISUALIZATION

// ---- VISUs/Visu_Stand.TcVIS
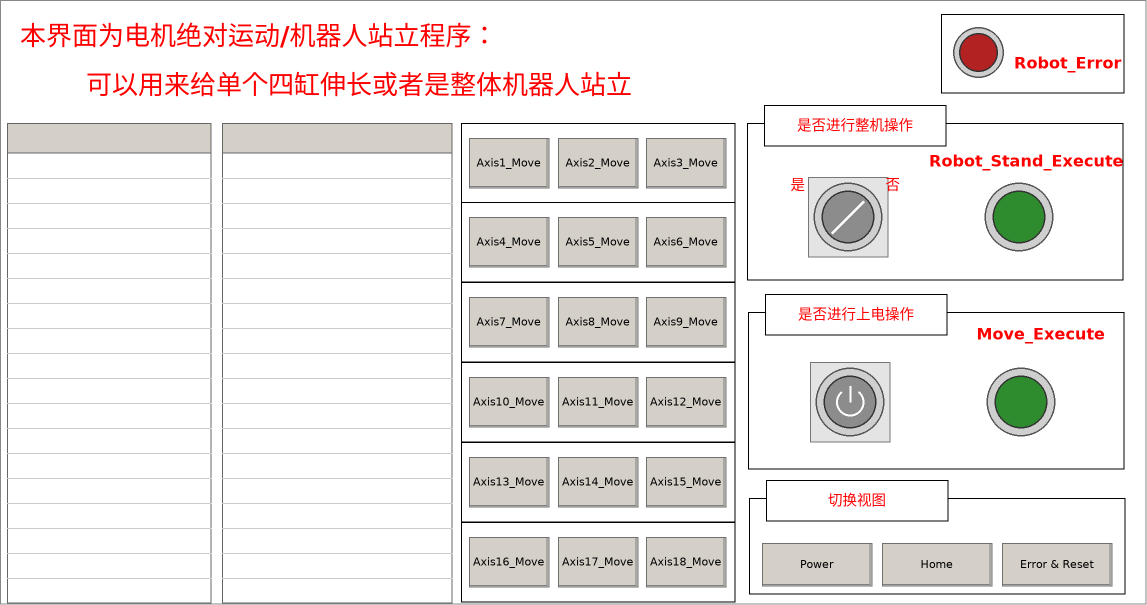
VISUALIZATION Visu_Stand  // 1147x605
    Rectangle (941,14 183x79)
    Rectangle (748,312 376x157)
    Label (964,318 154x32), "Move_Execute"
    Rectangle (765,294 182x41), "是否进行上电操作"
    Lamp1 (981,362 80x80), variable: MAIN.Move_Execute, style: Lamp-Lamp1-Green
    PowerSwitch (810,362 80x80), variable: MAIN.Move_Execute, behaviour: TOGGLE, style: Switch-PowerSwitch-Gray
    Lamp1 (948,23 61x59), variable: MAIN.Robot_Error, style: Lamp-Lamp1-Red
    Label (17,15 597x42), "本界面为电机绝对运动/机器人站立程序："
    Label (83,64 719x42), "可以用来给单个四缸伸长或者是整体机器人站立"
    Rectangle (747,123 376x157)
    Rectangle (764,105 182x41), "是否进行整机操作"
    Lamp1 (979,177 80x80), variable: MAIN.Robot_Stand_Execute, style: Lamp-Lamp1-Green
    RotarySwitch (808,177 80x80), variable: MAIN.Robot_Stand_Execute, behaviour: TOGGLE, style: Switch-RotarySwitch-Gray
    Label (863,170 60x30), "否"
    Label (768,170 60x30), "是"
    Label (991,47 154x32), "Robot_Error"
    Table (7,123 204x480), data array: MAIN.Axis_ActPostion
        p3854506369: MAIN.Axis_ActPostion[INDEX]
    Table (222,123 230x480), data array: MAIN.MoveAbsoluteDone
        p3854506369: MAIN.MoveAbsoluteDone[INDEX]
    Rectangle (461,123 274x80)
    Button (469,138 80x50), "Axis1_Move"
        toggle MAIN.Axis_Absolute_Eable[1]
    Button (646,138 80x50), "Axis3_Move"
        toggle MAIN.Axis_Absolute_Eable[3]
    Button (558,138 80x50), "Axis2_Move"
        toggle MAIN.Axis_Absolute_Eable[2]
    Rectangle (461,202 274x80)
    Button (469,217 80x50), "Axis4_Move"
        toggle MAIN.Axis_Absolute_Eable[4]
    Button (646,217 80x50), "Axis6_Move"
        toggle MAIN.Axis_Absolute_Eable[6]
    Button (558,217 80x50), "Axis5_Move"
        toggle MAIN.Axis_Absolute_Eable[5]
    Rectangle (461,282 274x80)
    Button (469,297 80x50), "Axis7_Move"
        toggle MAIN.Axis_Absolute_Eable[7]
    Button (646,297 80x50), "Axis9_Move"
        toggle MAIN.Axis_Absolute_Eable[9]
    Button (558,297 80x50), "Axis8_Move"
        toggle MAIN.Axis_Absolute_Eable[8]
    Rectangle (461,362 274x80)
    Button (469,377 80x50), "Axis10_Move"
        toggle MAIN.Axis_Absolute_Eable[10]
    Button (646,377 80x50), "Axis12_Move"
        toggle MAIN.Axis_Absolute_Eable[12]
    Button (558,377 80x50), "Axis11_Move"
        toggle MAIN.Axis_Absolute_Eable[11]
    Rectangle (461,442 274x80)
    Button (469,457 80x50), "Axis13_Move"
        toggle MAIN.Axis_Absolute_Eable[13]
    Button (646,457 80x50), "Axis15_Move"
        toggle MAIN.Axis_Absolute_Eable[15]
    Button (558,457 80x50), "Axis14_Move"
        toggle MAIN.Axis_Absolute_Eable[14]
    Rectangle (461,522 274x80)
    Button (469,537 80x50), "Axis16_Move"
        toggle MAIN.Axis_Absolute_Eable[16]
    Button (646,537 80x50), "Axis18_Move"
        toggle MAIN.Axis_Absolute_Eable[18]
    Button (558,537 80x50), "Axis17_Move"
        toggle MAIN.Axis_Absolute_Eable[17]
    Label (923,145 207x32), "Robot_Stand_Execute"
    Rectangle (749,498 376x96)
    Rectangle (766,480 182x41), "切换视图"
    Button (762,543 110x43), "Power"
        OnMouseClick: change screen: Visu_Power
    Button (1002,543 110x43), "Error & Reset"
        OnMouseClick: change screen: Visu_Reset
    Button (882,543 110x43), "Home"
        OnMouseClick: change screen: Visu_Home
END_VISUALIZATION
